// TIA Portal V15.1 export
// export: Created 2022-12-20T09:13:23.5739968Z, ExportSetting None, DisplayName Totally Integrated Automation Portal, DisplayVersion V15.1 Update 1, DisplayName TIA Portal Openness, DisplayVersion V15.1, DisplayName SINAMICS Startdrive Advanced, DisplayVersion V15.1, DisplayName G130, G150, S120, S150, SINAMICS MV, S210, DisplayVersion V15.1, DisplayName G110M, G120, G120C, G120D, G120P, DisplayVersion V15.1, DisplayName STEP 7 Professional, DisplayVersion V15.1 Update 1, DisplayName STEP 7 Safety, DisplayVersion V15.1, DisplayName WinCC Professional, DisplayVersion V15.1 Update 1, DisplayName SIMATIC Visualization Architect, DisplayVersion V15.1
FUNCTION_BLOCK "PLC_ESTOP_FB"   // FB511, LAD
TITLE = PLC ESTOP FB
{ S7_Optimized_Access := 'TRUE' }
// The block is used to control the Estops that switch off the complete line
// stored: AutoNumber false, MemoryReserve 100, SetENOAutomatically False
   VAR
      "000-AS01" : "CM_Estop_FB";   // Emergency stop HMI main 1 xxxx
   END_VAR
BEGIN

REGION Network 1: Call emergency stop HMI main 1 (AS01)
   // E-stop on main HMI
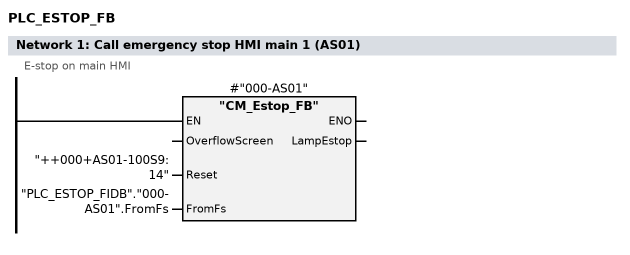
   RUNG wire#powerrail
      #"000-AS01"(OverflowScreen :=, Reset := "++000+AS01-100S9:14", FromFs := "PLC_ESTOP_FIDB"."000-AS01".FromFs, LampEstop =>)
   END_RUNG
   // the same network as SCL:
   #"000-AS01"(Reset := "++000+AS01-100S9:14", FromFs := "PLC_ESTOP_FIDB"."000-AS01".FromFs);   // "CM_Estop_FB"
END_REGION
END_FUNCTION_BLOCK
